// TIA Portal V19 export
FUNCTION_BLOCK "Block_2"   // FB1, SCL
{ S7_Optimized_Access := 'TRUE' }
// stored: MemoryReserve 100, SetENOAutomatically false
BEGIN
   IF TRUE THEN
       // Statement section IF
       ;
   END_IF;
END_FUNCTION_BLOCK
